{attribute 'GeneratedUsingTerminal: ELX5151-0000-0016'}
{attribute addProperty BoxType "ELX5151-0000-0016"}
{attribute addProperty Id "ENC_Status_compactAT %I*ENC_Status_compact_BFB16BB410ENC_Control_compactAT %Q*ENC_Control_compact_2ED727EF3WcStateAT %I*WcState_9091E0EB2InfoDataAT %I*InfoData_94A18F5E2"}
{attribute addProperty CRC "1870832292"}
{attribute addProperty Size "17"}
TYPE ELX5151_6F82A2A4 EXTENDS EtcSlaveTerminalBase_947E5A46 :
STRUCT
	{attribute addProperty Name "ENC_Status_compact"}
	ENC_Status_compact : ENC_Status_compact_BFB16BB4;
	{attribute addProperty Name "ENC_Control_compact"}
	ENC_Control_compact : ENC_Control_compact_2ED727EF;
	{attribute addProperty Name "WcState"}
	WcState : WcState_9091E0EB;
	{attribute addProperty Name "InfoData"}
	InfoData : InfoData_94A18F5E;
END_STRUCT
END_TYPE

(* stored: Version 1.2.0.0, ProductVersion 3.1.4024.9
   DUT ELX5151_6F82A2A4: Id {7b1bff27-50e4-41c0-904e-811bc8e2f5b6} *)
